TEXTLIST TextList_Infos
  0 = 'Langue' | FR: 'Langue' | EN: 'Language'
  1 = 'Id' | FR: 'Affaire :' | EN: 'Id:'
  2 = 'Auteur' | FR: 'Auteur :' | EN: 'Author:'
  3 = 'version' | FR: 'Version :' | EN: 'Release:'
  4 = 'date' | FR: 'Date :' | EN: 'Date:'
  5 = 'num' | FR: 'N° de série :' | EN: 'Serial number:'
  6 = 'type' | FR: 'Modèle :' | EN: 'Type:'
   = ''
END_TEXTLIST

(* stored: Version 1.1.0.1, ProductVersion 3.1.4024.10
   TextList TextList_Infos: Id {ab051693-5c79-499b-a5a8-016713a99840} *)
